{attribute addProperty BoxType "EP9128-0020-0016"}
{attribute addProperty Id "A_0004_EP9128_0021_0016A_0004_EP9128_0021_0016_5222794D4712589A_0001_EP9128_0020_0016_2_EP9128_1020EP9128_179A0949162A_0001_EP9128_0020_0016_3_EP9128_2020EP9128_179A0949162"}
{attribute addProperty CRC "2284188505"}
{attribute addProperty SizeInBites "4744"}
{attribute addProperty SizeInBytes "593"}
TYPE A_0001_EP9128_0020_0016_8825F359 EXTENDS EP9128_179A0949 :
STRUCT
	{attribute addProperty Name "A_0004_EP9128_0021_0016"}
	A_0004_EP9128_0021_0016 : A_0004_EP9128_0021_0016_5222794D;
	{attribute addProperty Name "A_0001_EP9128_0020_0016_2_EP9128_1020"}
	A_0001_EP9128_0020_0016_2_EP9128_1020 : EP9128_179A0949;
	{attribute addProperty Name "A_0001_EP9128_0020_0016_3_EP9128_2020"}
	A_0001_EP9128_0020_0016_3_EP9128_2020 : EP9128_179A0949;
END_STRUCT
END_TYPE

(* stored: Version 1.2.0.0, ProductVersion 3.1.4024.9
   DUT A_0001_EP9128_0020_0016_8825F359: Id {6bcdb496-5735-4890-a1bc-c99926ec5473} *)
